{attribute 'qualified_only'}
{attribute 'strict'}
{attribute 'to_string'}
TYPE AxisMotionState :
(
    Undefined,
    Disabled,
    Standstill,
    ErrorStop,
    Stopping,
    Homing,
    DiscreteMotion,
    ContinuousMotion,
    SynchronisedMotion
);
END_TYPE

(* stored: Version 1.1.0.1
   DUT AxisMotionState: Id {77000085-24a7-49b6-b20b-f782d4e0ef83} *)
